TYPE Astrofan612FfuEvent :
STRUCT
	ThresholdPercent : UINT;
	TimerSeconds : UINT;
END_STRUCT
END_TYPE

(* stored: Version 1.1.0.1, ProductVersion 3.1.4024.12
   DUT Astrofan612FfuEvent: Id {6fab683f-7259-4d6f-b102-faa964c934a5} *)
